// TIA Portal V17 export
// export: Created 2024-09-02T12:49:57.1862692Z, ExportSetting WithDefaults, DisplayName Totally Integrated Automation Portal, DisplayVersion V17, DisplayName TIA Portal Openness, DisplayVersion V17, DisplayName TIA Portal Version Control Interface, DisplayVersion V17, DisplayName STEP 7 Professional, DisplayVersion V17, DisplayName STEP 7 Safety, DisplayVersion V17, DisplayName WinCC Professional, DisplayVersion V17
DATA_BLOCK "SysDB_PNIO_DiagDetail"   // DB1296
{ S7_Optimized_Access := 'TRUE'; DB_Accessible_From_OPC_UA := 'FALSE' }
AUTHOR : OlegFuehrus
FAMILY : DIAG
NAME : DIAG
VERSION : 0.1
// stored: AutoNumber true, DBAccessibleFromOPCUA false, IsOnlyStoredInLoadMemory false, IsRetainMemResEnabled false, IsWriteProtectedInAS false, MemoryReserve 0
   VAR
      "Checking active" : Bool;
      Profinet_Disturbed : Bool;
      Profinet_Fault : Bool;
      Failed : Int;
      Disturbance : Int;
      First_Executed : Int;
      First_Disturbed : Int;
      Report_Slave : Array[0..1023] of Bool;
      Slaves_Available : Array[0..1023] of Bool;
      Slaves_Configured : Array[0..1023] of Bool;
      Slaves_Disturbed : Array[0..1023] of Bool;
      Slaves_Deactivated : Array[0..1023] of Bool;
   END_VAR
BEGIN
END_DATA_BLOCK
